FUNCTION F_UDINT_TO_DINT : DINT
VAR_INPUT
    value : UDINT;
END_VAR
VAR
    inRangeValue : UDINT;
END_VAR

IF value.31 THEN // out of range
    F_Assert(
        Assertion := FALSE,
        FailMessage := 'Input arg of F_UDINT_TO_DINT too large to convert, so value of Max DINT (2147483647) was returned');

    inRangeValue := 16#7FFF_FFFF; // ‭Max DINT = 2147483647‬
ELSE
    inRangeValue := value;
END_IF
F_UDINT_TO_DINT := UDINT_TO_DINT(inRangeValue);

END_FUNCTION

(* stored: Version 1.1.0.1, ProductVersion 3.1.4024.3
   POU F_UDINT_TO_DINT: Id {385cda2d-2d58-4cf8-a0cc-93acc0027c7b}, SpecialFunc None *)
